# B&R Automation Studio project PLCEksamen1
Automation Studio 4.5.2.102

## Configuration Config1

### Hardware
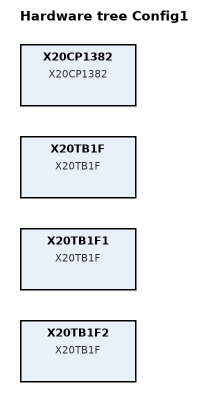
```
X20CP1382 : X20CP1382 v1.7.0.0  [X1 -> X1.SL; X2 -> X2.SL; X3 -> X3.SL]
  Module X1 (Type=X1, Virtual=true, Version=1.7.0.0)
    Connection (Connector=SS1, TargetModule=X20TB1F, TargetConnector=SS)
    Connection (Connector=SL, TargetModule=X20CP1382, TargetConnector=X1)
  Module X2 (Type=X2, Virtual=true, Version=1.7.0.0)
    Connection (Connector=SS1, TargetModule=X20TB1F1, TargetConnector=SS)
    Connection (Connector=SL, TargetModule=X20CP1382, TargetConnector=X2)
  Module X3 (Type=X3, Virtual=true, Version=1.7.0.0)
    Connection (Connector=SS1, TargetModule=X20TB1F2, TargetConnector=SS)
    Connection (Connector=SL, TargetModule=X20CP1382, TargetConnector=X3)
  Connector IF2:
    ActivateDevice = 1
  ConfigurationID = PLCEksamen_Config1
X20TB1F : X20TB1F v1.0.0.0
X20TB1F1 : X20TB1F v1.0.0.0
X20TB1F2 : X20TB1F v1.0.0.0
```

## Logical view

Binary libraries used (declarations not repeated): operator, runtime, astime, AsIecCon, standard

### Program Logical/Program

#### Variables.var
```iecst
VAR
	diPos2OutOfPlace : BOOL;
	diPos1OutOfPlace : BOOL;
	diPos1OutOfPlaceWeight: INT;
	diPos2OutOfPlaceWeight: INT;
	doGoBtn : BOOL;
	doConvMainStart : BOOL;
	ConvMainStop : BOOL;
	doRobotToPos2 : BOOL;
	doRobotToPos1 : BOOL;
	pickerRobotRight : RobotArm;
	pickerRobotLeft : RobotArm;
	SorterRobot : RobotArm;
	diConvSideRunning : BOOL;
	diConvMainRunning : BOOL;
	diRightPos : BOOL;
	diWeightScale: WORD;
	toPicker : F_TRIG;
	rightTrig: F_TRIG;
	leftTrig: F_TRIG;
	diDeliveryTrigRight : F_TRIG;
	diDeliveryTrigLeft : F_TRIG;
	diPickingSensor : BOOL;
	toBePicked : USINT;
	doStackerRight : BOOL;
	doStackerLeft : BOOL;
	doStackerPick : BOOL;
	doSorterPick : BOOL;
	doConvSideStart : BOOL;
	diConvSideStop : BOOL;
	doFeederMid : BOOL;
	doFeederLeft : BOOL;
	doFeederRight : BOOL;
	FeedCount : USINT;
	Stacked : BOOL;
	stackingTrig : R_TRIG;
	Timer : TON;
	SorterTimer : TON;
	StackerTimer : TON;

	TimerSideConv: TON;
END_VAR
```

#### Main.st
```iecst
PROGRAM _INIT
	(* Init værdier for alt i programmet *)

	doGoBtn := FALSE; // input fra experior
	diPos1OutOfPlace := FALSE; // input fra experior weight 1
	diPos2OutOfPlace := FALSE; // input fra experior weight 2
	diConvMainRunning := FALSE; // input fra experior om bånd status på hovedbånd
	diConvSideRunning := FALSE; // input fra experior om bånd status på afleverings bånd
	doConvMainStart := FALSE; // output til experior
	ConvMainStop := FALSE;
	doRobotToPos1 := FALSE; // output til robot
	doRobotToPos2 := FALSE; // output til robot
	Timer.PT := T#3s;
	TimerSideConv.PT := T#4s;
	SorterTimer.PT := T#0.5s;
	StackerTimer.PT := T#1s;
END_PROGRAM

PROGRAM _CYCLIC
	(* Go knappen som starter hele programmet*)
	IF doGoBtn = TRUE AND ConvMainStop = FALSE THEN
		doConvMainStart := TRUE;
		Timer.IN := TRUE;

	ELSIF doGoBtn = TRUE AND ConvMainStop = TRUE THEN
		doConvMainStart := FALSE;
		Timer.IN := FALSE;

	ELSIF doGoBtn = FALSE AND ConvMainStop = TRUE THEN
		ConvMainStop := FALSE;
		doConvMainStart := FALSE;

	ELSE
		ConvMainStop := TRUE;
		Timer.IN := FALSE;
	END_IF;
	(*Hvis der trykkes stop eller bliver sendt stop signal skal båndet stoppe.*)
	//IF diConvMainStop = TRUE THEN
	//diConvMainStart := FALSE;
	//diConvMainStop := FALSE;
	//END_IF;

	IF diWeightScale > 300 AND doGoBtn = TRUE THEN
		SorterTimer.IN := TRUE;
		IF SorterTimer.Q THEN
			doSorterPick := TRUE;
			SorterTimer.IN := FALSE;
		END_IF;
	ELSE
		SorterTimer.IN := FALSE;
		doSorterPick := FALSE;
	END_IF;
(*	IF diConvMainRunning = TRUE AND diPos1OutOfPlaceWeight = TRUE AND diPos2OutOfPlaceWeight = FALSE THEN
		doRobotToPos1 := TRUE;
		doSorterPick := TRUE;
	ELSE
		doRobotToPos1 := FALSE;
	END_IF;
	IF diConvMainRunning = TRUE AND diPos2OutOfPlace = TRUE AND diPos1OutOfPlace = FALSE THEN
		doRobotToPos2 := TRUE;
		doSorterPick := TRUE;
	ELSE
		doRobotToPos2 := FALSE;
	END_IF;
	IF diConvMainRunning = TRUE AND diPos2OutOfPlace = TRUE AND diPos1OutOfPlace = TRUE THEN
		ConvMainStop := TRUE;
		doRobotToPos1 := TRUE;
		doSorterPick := TRUE;

		IF SorterRobot.Delivering = TRUE THEN
			doRobotToPos1 := FALSE;
			doRobotToPos2 := TRUE;
			SorterRobot.Delivering := FALSE;

			IF SorterRobot.Delivering = TRUE THEN
				doRobotToPos2 := FALSE;
				ConvMainStop := FALSE;
			END_IF;

		END_IF;

	END_IF; *)
	// denne IF sætning styrer fodning af kasser. tæller op til 2, går derefter ned til 0 igen og starter forfra. stiger 1 hver gang Timer.Q pulser.
	IF FeedCount = 0 AND Timer.Q THEN
		doFeederLeft := TRUE;
		doFeederRight := FALSE;
		FeedCount := FeedCount+1;
		Timer.IN := FALSE;
	ELSIF FeedCount = 1 AND Timer.Q THEN
		doFeederMid := TRUE;
		doFeederLeft := FALSE;
		FeedCount := FeedCount+1;
		Timer.IN := FALSE;
	ELSIF FeedCount = 2 AND Timer.Q THEN
		doFeederRight := TRUE;
		doFeederMid := FALSE;
		Timer.IN := FALSE;
		FeedCount := 0;
	END_IF;
	//stacker kontrol kode
	IF toPicker.Q THEN
		toBePicked := toBePicked+1;
	END_IF;

	IF toBePicked >= 1 THEN
		StackerTimer.IN := TRUE;
		IF StackerTimer.Q THEN
			doStackerPick := TRUE;
			StackerTimer.IN := FALSE;
		END_IF;
	ELSE
		StackerTimer.IN := FALSE;
		doStackerPick := FALSE;
	END_IF;
	IF toBePicked <= 1 AND leftTrig.Q THEN

		toBePicked := toBePicked-1;
	ELSIF toBePicked >= 1 AND rightTrig.Q THEN
		toBePicked := toBePicked-1;
	END_IF;
	IF stackingTrig.Q THEN
		doConvSideStart := TRUE;
		TimerSideConv.IN := TRUE;
	ELSIF diConvSideRunning = TRUE AND TimerSideConv.Q THEN
		doConvSideStart := FALSE;
		TimerSideConv.IN := FALSE;
	END_IF;

	TimerSideConv();
	Timer();
	toPicker(CLK := diPickingSensor);
	stackingTrig(CLK := Stacked);
	rightTrig (CLK := pickerRobotRight.Getting);
	leftTrig (CLK := pickerRobotLeft.Getting);
	SorterTimer();
	StackerTimer();
			END_PROGRAM

			PROGRAM _EXIT
			(* Insert code here *)

			END_PROGRAM
```
